(* PLC project PLC, Beckhoff Automation GmbH TwinCAT PLC Control 3.5.13.21 *)
(* stored: creationDateTime 2024-02-17T22:42:25.5394115, modificationDateTime 2024-02-17T22:42:25.5394115 *)

TYPE LPOutput :
STRUCT
	on AT %Q*: BOOL;
END_STRUCT
END_TYPE
